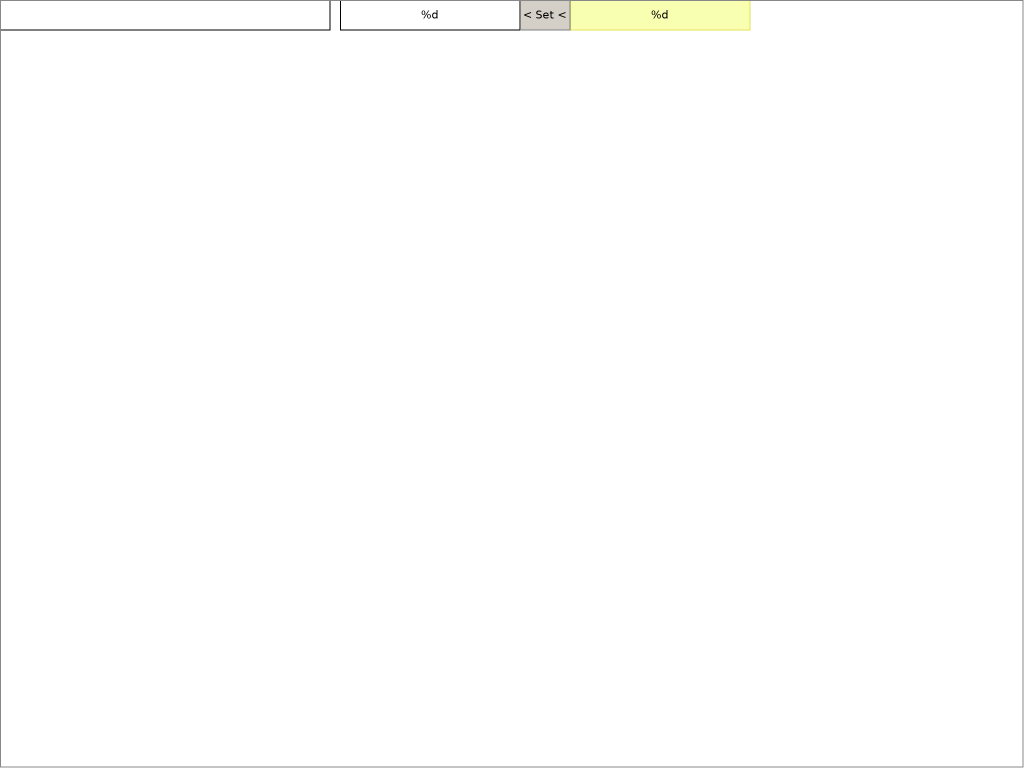
VISUALIZATION Param_DINT  // 1024x768
VAR_INPUT
	nIdx:		INT;
END_VAR
    Rectangle (340,0 180x30), "%d", text variable: stMParam_Visu.nDintAktValue[nIdx]
    Rectangle (0,0 330x30), text list: 'TL_Params_INT', text index: nIdx
    Rectangle (570,0 180x30), "%d", text variable: stMParam_Visu.nDintNewValue[nIdx]
        OnMouseClick: write the text variable via Default
    Rectangle (520,0 50x30), "< Set <"
        OnMouseClick: execute { stMParam_Visu.bDintSetValue[nIdx]:=TRUE; }
END_VISUALIZATION

(* stored: Version 1.1.0.1, ProductVersion 3.1.4024.12
   Visu Param_DINT: Id {12e9932e-cca8-4d2d-91d7-1113188b3710} *)
